{attribute 'GeneratedUsingTerminal: AT2000-5233-0019'}
{attribute addProperty BoxType "AT2000-5233-0019"}
{attribute addProperty Description "AT2000-5233 Sensor line 233 mm"}
{attribute addProperty Physics "K"}
{attribute addProperty Id "FB_InputsAT %I*FB_Inputs_4BC4AA0166FB_OutputsAT %Q*FB_Outputs_DAFD38E02WcStateAT %I*WcState_9091E0EB2InfoDataAT %I*InfoData_A7436BC610"}
{attribute addProperty CRC "866377499"}
{attribute addProperty Size "80"}
TYPE AT2000_33A3DF1B EXTENDS EtcSlaveTerminalBase_947E5A46 :
STRUCT
	{attribute addProperty Name "FB_Inputs"}
	FB_Inputs : FB_Inputs_4BC4AA01;
	{attribute addProperty Name "FB_Outputs"}
	FB_Outputs : FB_Outputs_DAFD38E0;
	{attribute addProperty Name "WcState"}
	WcState : WcState_9091E0EB;
	{attribute addProperty Name "InfoData"}
	InfoData : InfoData_A7436BC6;
END_STRUCT
END_TYPE

(* stored: Version 1.2.0.0, ProductVersion 3.1.4024.11
   DUT AT2000_33A3DF1B: Id {426a42b0-cf33-406b-a6da-bc31144b8f8a} *)
